// TIA Portal V18 export
FUNCTION_BLOCK "Baustein_Int"   // FB2, FBD
{ S7_Optimized_Access := 'TRUE' }
// stored: MemoryReserve 100, SetENOAutomatically false
   VAR_INPUT
      Test_1 : Int := 120;
      Test_2 : Bool := true;
   END_VAR
   VAR_OUTPUT
      Output_1 : Int := 120;
      Output_2_1 : Int := 78;
      Output_2 : Bool := true;
   END_VAR
BEGIN
END_FUNCTION_BLOCK
